KUKA KRL program: chk_w3_grp5_opn.src

&ACCESS RVO1
&COMMENT Check GRP Z5 ACTROS OPEN
DEF chk_w3_grp5_opn( )

; Check gripper actros OPEN Z5
;//---- Start User-------

$TIMER[10] = 0
$TIMER_STOP[10] = FALSE

WAIT FOR (NOT $IN[28])
WAIT FOR ($IN[27])

$TIMER_STOP[10] = TRUE
$TIMER[10] = 0

;//---- End User---------

END
